TYPE ST_ServoStatus :
STRUCT
	
	//Status : AXIS_REF.Status;

END_STRUCT
END_TYPE

(* stored: Version 1.1.0.1, ProductVersion 3.1.4024.12
   DUT ST_ServoStatus: Id {feaef20d-4570-406d-a8e3-4d5690e10e6d} *)
